// TIA Portal V17 export
// export: Created 2022-03-18T16:55:07.1321486Z, ExportSetting WithDefaults, DisplayName Totally Integrated Automation Portal, DisplayVersion V17, DisplayName TIA Portal Openness, DisplayVersion V17, DisplayName TIA Portal Version Control Interface, DisplayVersion V17, DisplayName SINAMICS Startdrive Advanced, DisplayVersion V17, DisplayName SINAMICS Startdrive G130, G150, S120, S150, SINAMICS MV, S210, DisplayVersion V17, DisplayName SINAMICS Startdrive G110M, G120, G120C, G120D, G120P, G115D, DisplayVersion V17, DisplayName STEP 7 Professional, DisplayVersion V17, DisplayName STEP 7 Safety, DisplayVersion V17, DisplayName WinCC Advanced / Unified PC, DisplayVersion V17
ORGANIZATION_BLOCK "Main"   // OB1, LAD, ProgramCycle
TITLE = "Main Program Sweep (Cycle)"
{ S7_Optimized_Access := 'TRUE' }
VERSION : 0.1
// stored: AutoNumber true, IsIECCheckEnabled false, SetENOAutomatically false
   VAR_INPUT
      Initial_Call : Bool;   // Initial call of this OB
      Remanence : Bool;   // =True, if remanent data are available
   END_VAR
BEGIN

REGION Network 1 (SCL): test velocità lettura dati
   // "M1_out".sp_speed := "M1_out".sp_speed + 1;
   // IF "M1_out".sp_speed > 10000 THEN
   //     "M1_out".sp_speed := 0;
   // END_IF;

   // "M1_out".sp_acc := "M1_out".sp_acc + 1;
   // IF "M1_out".sp_acc > 10000 THEN
   //     "M1_out".sp_acc := 0;
   // END_IF;
END_REGION

REGION Network 2 (SCL): Motore 1
   "M1_instance_DB"(M_in := "M1_in",
                    M_out => "M1_out");


   "instance_ciclo_mac"();
END_REGION
END_ORGANIZATION_BLOCK
